// TIA Portal V20 export
ORGANIZATION_BLOCK "Main"   // OB1, LAD, ProgramCycle
TITLE = "Main Program Sweep (Cycle)"
{ S7_Optimized_Access := 'TRUE' }
// stored: SetENOAutomatically false
   VAR_INPUT
      Initial_Call : Bool;   // Initial call of this OB
      Remanence : Bool;   // =True, if remanent data are available
   END_VAR
BEGIN

REGION Network 1 (SCL)
   "SynchronousAxisCam_DB"(Start:= "STSRT_",
                             synchronousAxisCamRef_1:= "SynchronousAxis_1",
                             synchronousAxisCamRef_2:= "SynchronousAxis_2",
                             virtualAxisRef:= "virtual _master_axis",
                             camRef:= "Cam_1");
END_REGION
END_ORGANIZATION_BLOCK
